TYPE ST_ESDStep :
STRUCT
	sDescription    : STRING;       // what this step does
    tTimeout        : TIME;         // max time allowed
    bComplete       : BOOL;         // step confirmed done
    bFailed         : BOOL;         // step timed out
END_STRUCT
END_TYPE

(* stored: Version 1.1.0.1, ProductVersion 3.1.4024.16
   DUT ST_ESDStep: Id {f837d3a1-cead-4e0a-92d3-c364e601357f} *)
